Staubli VAL3: bDialogYesNo.pgx

public program bDialogYesNo(string x_sTitle, string x_sQuestion_r1, string x_sQuestion_r2, string x_sQuestion_r3, bool& x_bResp)
  local bool l_bLoop
  local num l_nNum
begin

  //return by using the bResp parameter true if the choose was "yes", false if the choose was "no"
  //notes: screen size is 13rowsX40columns
  //usage: call bDialogYesNo(bRes, "RETURN IN HOME", "ATTENTION:", "Robot will return in home position", "continue?")

  wait(getKey()==-1)

  userPage()
  call clrscr()

  call sCenterTitle(x_sTitle)

  title(x_sTitle)

  gotoxy(0,4)
  call sCenterRow(x_sQuestion_r1)
  putln(x_sQuestion_r1)

  gotoxy(0,5)
  call sCenterRow(x_sQuestion_r2)
  putln(x_sQuestion_r2)

  gotoxy(0,6)
  call sCenterRow(x_sQuestion_r3)
  putln(x_sQuestion_r3)

  gotoxy(0,13)
  put("F1=No")
  gotoxy(34,13)
  put("F8=Yes")

  do
    l_nNum=get()
    if l_nNum==271
      x_bResp=false
    elseIf l_nNum==278
      x_bResp=true
    endIf
  until l_nNum==271 or l_nNum==278

  call clrscr()

  wait(getKey()==-1)

end
